Yaskawa INFORM job: TWIN_FRONT_SEARCH_90ST-1_5340.JBI

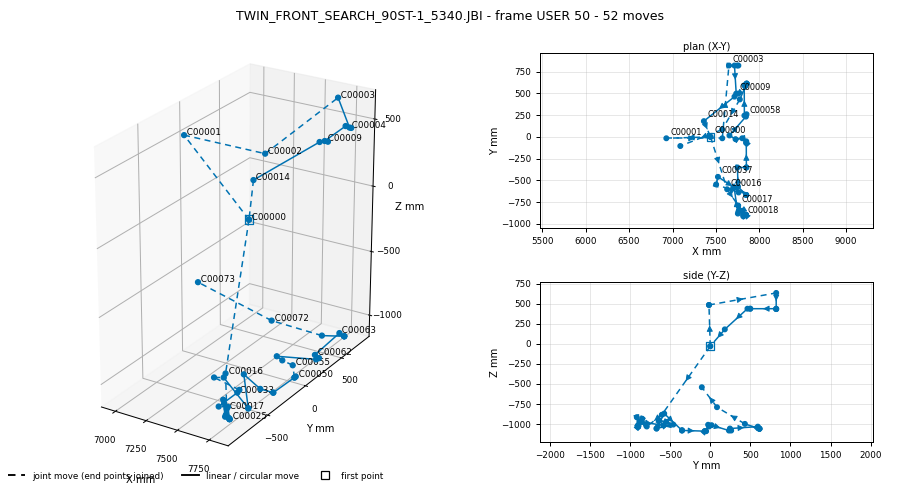
[picture p0: tool path of TWIN_FRONT_SEARCH_90ST-1_5340.JBI in frame USER 50, 52 of 56 moves have a stored position in this frame; points joined in program order, loops and branches not executed]
/JOB
//NAME TWIN_FRONT_SEARCH_90ST-1_5340
///FOLDERNAME 02-SKRZYNIE_JOBS
//POS
///NPOS 74,74,0,10,0,0
///USER 50
///TOOL 0
///POSTYPE USER
///RECTAN
///RCONF 0,0,1,0,0,0,0,0,0,0,0,0,0,0,0,0,0,0,0,0,0,0,0,0
C00000=7437.393,0.308,-30.113,-0.0036,-53.6521,0.0034
///RCONF 1,0,1,0,0,0,0,0,0,0,0,0,0,0,0,0,0,0,0,0,0,0,0,0
C00001=6928.400,-15.669,483.666,2.7707,-42.5282,-1.8493
C00002=7572.625,-15.669,483.666,2.7707,-42.5282,-1.8493
C00003=7649.331,821.904,633.544,31.3308,-50.3097,5.8371
C00004=7744.036,821.924,432.600,31.3309,-50.3106,5.8382
C00005=7764.657,821.900,432.619,31.3298,-50.3131,5.8368
C00006=7758.075,821.902,432.614,31.3294,-50.3128,5.8375
C00007=7758.087,821.893,399.298,31.3287,-50.3132,5.8373
C00008=7713.156,821.903,437.297,31.3290,-50.3132,5.8374
C00009=7733.152,498.705,437.301,28.5621,-56.7278,8.0159
C00010=7764.512,498.715,437.279,28.5577,-56.7277,8.0212
C00011=7758.151,498.718,437.279,28.5586,-56.7273,8.0207
C00012=7758.152,498.721,398.863,28.5594,-56.7235,8.0206
C00013=7713.145,463.670,437.302,31.3284,-50.3136,5.8380
C00014=7360.642,181.544,179.903,-30.3084,-22.7119,47.7634
///RCONF 0,0,1,0,0,0,0,0,0,0,0,0,0,0,0,0,0,0,0,0,0,0,0,0
C00015=7437.393,0.308,-30.113,-0.0036,-53.6521,0.0034
///RCONF 0,0,0,0,0,0,0,0,0,0,0,0,0,0,0,0,0,0,0,0,0,0,0,0
C00016=7628.865,-602.935,-884.155,-14.6080,-23.9960,-22.0349
///RCONF 1,0,0,0,0,0,0,0,0,0,0,0,0,0,0,0,0,0,0,0,0,0,0,0
C00017=7755.981,-790.379,-1030.058,-1.3034,-14.2488,-53.7856
C00018=7814.982,-914.673,-915.183,-49.7301,36.0224,40.1931
C00019=7814.976,-893.416,-1010.060,-49.7313,36.0195,40.1889
C00020=7814.973,-903.090,-1020.024,-49.7309,36.0192,40.1886
C00021=7814.980,-919.884,-1020.010,-49.7305,36.0200,40.1893
///RCONF 0,0,0,0,0,0,0,0,0,0,0,0,0,0,0,0,0,0,0,0,0,0,0,0
C00022=7765.216,-847.521,-933.099,-41.9556,-3.8768,2.5162
C00023=7838.256,-897.742,-1022.780,33.2636,-28.1441,-95.3546
C00024=7838.227,-897.761,-1034.874,33.2614,-28.1452,-95.3536
C00025=7845.758,-897.726,-1031.582,33.2648,-28.1427,-95.3555
C00026=7845.758,-897.726,-1031.582,33.2648,-28.1427,-95.3555
C00027=7845.758,-897.726,-1031.582,33.2648,-28.1427,-95.3555
C00028=7845.758,-897.726,-1031.582,33.2648,-28.1427,-95.3555
C00029=7863.986,-897.727,-1031.592,33.2632,-28.1430,-95.3545
C00030=7803.420,-850.217,-974.308,33.2648,-28.1422,-95.3567
///RCONF 1,0,0,0,0,0,0,0,0,0,0,0,0,0,0,0,0,0,0,0,0,0,0,0
C00031=7813.345,-897.089,-897.203,54.9948,73.9690,-177.4313
C00032=7752.242,-882.487,-971.733,-38.0360,-24.7001,-17.6899
C00033=7709.308,-583.044,-1014.454,-8.5802,-15.4711,-34.3684
///RCONF 0,0,0,0,0,0,0,0,0,0,0,0,0,0,0,0,0,0,0,0,0,0,0,0
C00034=7760.363,-639.479,-954.196,-16.2283,58.5864,108.1042
///RCONF 1,0,0,0,0,0,0,0,0,0,0,0,0,0,0,0,0,0,0,0,0,0,0,0
C00035=7501.819,-547.461,-973.110,-40.0484,29.0713,48.7679
C00036=7849.163,-652.269,-1055.293,-36.7283,45.9336,63.6180
C00037=7522.707,-459.746,-1006.152,21.9891,-7.6328,-78.4767
///RCONF 0,0,0,0,0,0,0,0,0,0,0,0,0,0,0,0,0,0,0,0,0,0,0,0
C00038=7848.448,-668.635,-1055.276,-38.1211,38.1551,84.2772
C00039=7848.418,-668.637,-1070.622,-38.1202,38.1533,84.2760
C00040=7859.950,-668.642,-1067.637,-38.1207,38.1516,84.2738
C00041=7848.448,-668.635,-1055.276,-38.1211,38.1551,84.2772
///RCONF 1,0,0,0,0,0,0,0,0,0,0,0,0,0,0,0,0,0,0,0,0,0,0,0
C00042=7753.744,-572.921,-869.370,35.5853,8.2503,-84.4804
///RCONF 0,0,0,0,0,0,0,0,0,0,0,0,0,0,0,0,0,0,0,0,0,0,0,0
C00043=7760.219,-665.415,-840.606,-36.5266,43.0988,92.6871
C00044=7778.037,-351.548,-1078.962,-31.8373,42.1277,84.4329
C00045=7747.357,-351.554,-1078.963,-31.8382,42.1272,84.4305
///RCONF 1,0,0,0,0,0,0,0,0,0,0,0,0,0,0,0,0,0,0,0,0,0,0,0
C00046=7850.194,-351.548,-1078.962,-31.8375,42.1274,84.4323
C00047=7850.215,-351.581,-1093.915,-31.8403,42.1281,84.4282
C00048=7861.111,-351.581,-1090.949,-31.8408,42.1244,84.4218
C00049=7850.194,-351.548,-1078.962,-31.8375,42.1274,84.4323
C00050=7848.886,-51.045,-1088.766,-31.8328,42.1278,99.9917
C00051=7848.894,-68.663,-1088.753,-31.8329,42.1298,99.9929
C00052=7848.906,-68.683,-1101.493,-31.8343,42.1324,99.9922
C00053=7861.752,-68.689,-1098.467,-31.8340,42.1361,99.9970
C00054=7848.894,-68.663,-1088.753,-31.8329,42.1298,99.9929
C00055=7802.761,-15.645,-1029.914,-9.7407,56.5457,162.3768
///RCONF 0,0,0,0,0,0,0,0,0,0,0,0,0,0,0,0,0,0,0,0,0,0,0,0
C00056=7725.278,-25.980,-1008.468,-14.6300,-10.2329,22.0522
C00057=7655.312,16.758,-1013.968,36.3468,26.5568,-107.0138
///RCONF 1,0,0,0,0,0,0,0,0,0,0,0,0,0,0,0,0,0,0,0,0,0,0,0
C00058=7844.634,233.760,-1080.855,23.4698,44.5725,-116.2756
C00059=7851.838,260.958,-1080.540,23.4723,44.5715,-116.2716
C00060=7851.821,261.021,-1099.017,23.4678,44.5749,-116.2769
C00061=7860.953,261.032,-1096.049,23.4627,44.5753,-116.2825
C00062=7827.288,245.626,-1055.543,23.4731,44.5712,-116.2696
C00063=7825.305,593.191,-1032.010,10.4642,52.1554,-131.8432
C00064=7853.529,612.933,-1058.080,10.4637,52.1549,-131.8455
C00065=7853.595,612.880,-1072.989,10.4677,52.1564,-131.8443
C00066=7853.565,612.921,-1058.045,10.4627,52.1566,-131.8492
C00067=7868.536,612.906,-1058.021,10.4653,52.1574,-131.8467
C00068=7853.558,612.926,-1058.047,12.0695,52.4631,-119.3669
C00069=7853.529,635.104,-1058.094,12.7425,52.9997,-118.8215
C00070=7853.561,612.917,-1058.050,10.4623,52.1563,-127.3651
C00071=7774.620,431.852,-997.566,17.4286,48.8596,-123.7766
C00072=7570.947,84.363,-789.769,8.3295,54.7414,-178.0447
C00073=7089.401,-104.773,-541.114,-34.6747,-14.1850,36.1511
///RCONF 0,0,0,0,0,0,0,0,0,0,0,0,0,0,0,0,0,0,0,0,0,0,0,0
BC00000=5622.975
BC00001=5622.975
BC00002=6267.199
BC00003=6480.663
BC00004=6480.663
BC00005=6480.663
BC00006=6480.663
BC00007=6480.663
BC00008=6480.663
BC00009=6480.663
BC00010=6480.663
BC00011=6480.663
BC00012=6480.663
BC00013=6480.663
BC00014=6140.736
BC00015=5622.975
BC00016=6179.171
BC00017=6446.713
BC00018=6446.759
BC00019=6446.759
BC00020=6446.759
BC00021=6446.759
BC00022=6446.759
BC00023=6446.759
BC00024=6446.759
BC00025=6446.759
BC00026=6446.759
BC00027=6446.759
BC00028=6446.759
BC00029=6446.759
BC00030=6446.759
BC00031=6446.759
BC00032=6446.759
BC00033=6379.471
BC00034=6379.472
BC00035=6162.623
BC00036=6515.049
BC00037=6162.623
BC00038=6515.049
BC00039=6515.049
BC00040=6515.049
BC00041=6515.049
BC00042=6419.547
BC00043=6419.547
BC00044=6442.892
BC00045=6445.014
BC00046=6515.049
BC00047=6515.049
BC00048=6515.049
BC00049=6515.049
BC00050=6515.049
BC00051=6515.049
BC00052=6515.049
BC00053=6515.049
BC00054=6515.049
BC00055=6439.422
BC00056=6439.422
BC00057=6307.353
BC00058=6515.049
BC00059=6515.049
BC00060=6515.049
BC00061=6515.049
BC00062=6515.049
BC00063=6515.029
BC00064=6515.029
BC00065=6515.035
BC00066=6515.035
BC00067=6515.035
BC00068=6515.035
BC00069=6515.035
BC00070=6515.035
BC00071=6515.035
BC00072=6132.885
BC00073=5388.459
///POSTYPE BASE
P00006=-2.449,0.031,8.825,0.0000,0.0000,0.0000
P00021=6.550,-0.003,-5.735,0.0000,0.0000,0.0000
P00022=5.943,-0.018,-6.388,0.0000,0.0000,0.0000
P00058=0.000,0.000,3.000,0.0000,0.0000,0.0000
///RCONF 1,0,0,0,0,0,0,0,0,0,0,0,0,0,0,0,0,0,0,0,0,0,0,0
P00500=2.332,-5.281,-1.258,0.0000,0.0000,0.0000
///RCONF 0,0,0,0,0,0,0,0,0,0,0,0,0,0,0,0,0,0,0,0,0,0,0,0
P00501=-2.026,0.009,3.534,0.0000,0.0000,0.0000
///RCONF 1,0,0,0,0,0,0,0,0,0,0,0,0,0,0,0,0,0,0,0,0,0,0,0
P00502=-2.023,0.001,1.732,0.0000,0.0000,0.0000
P00503=0.138,-0.044,1.539,0.0000,0.0000,0.0000
P00504=-0.309,-0.010,1.636,0.0000,0.0000,0.0000
P00505=0.999,-9.916,8.214,0.0000,0.0000,0.0000
//INST
///DATE 2025/01/21 12:44
///ATTR SC,RW,RJ
////FRAME USER 50
///GROUP1 RB1,BS1
NOP
MOVJ C00000 BC00000 VJ=50.00
MOVJ C00001 BC00001 VJ=50.00
MOVJ C00002 BC00002 VJ=50.00
MOVJ C00003 BC00003 VJ=50.00
MOVL C00004 BC00004 V=166.7
REFP 3 C00005 BC00005
CALL JOB:SEARCH-R1
SET P0021 P0006
SFTON P0021
MOVL C00006 BC00006 V=333.3 PL=0
REFP 3 C00007 BC00007
CALL JOB:SEARCH-R1
SET P0021 P0006
SFTON P0021
SFTOF
MOVL C00008 BC00008 V=166.7
MOVL C00009 BC00009 V=166.7
REFP 3 C00010 BC00010
CALL JOB:SEARCH-R1
SET P0022 P0006
SFTON P0022
MOVL C00011 BC00011 V=333.3 PL=0
REFP 3 C00012 BC00012
CALL JOB:SEARCH-R1
SET P0022 P0006
SFTON P0022
SFTOF
MOVL C00013 BC00013 V=166.7
MOVL C00014 BC00014 V=333.3
MOVJ C00015 BC00015 VJ=50.00
MOVJ C00016 BC00016 VJ=50.00
MOVJ C00017 BC00017 VJ=30.00
MOVJ C00018 BC00018 VJ=20.00
'::::::::::::::::::::::::::::::::
'W21 P
'::::::::::::::::::::::::::::::::
MOVL C00019 BC00019 V=500.0
MOVL C00020 BC00020 V=333.3 PL=0
REFP 3 C00021 BC00021
CALL JOB:SEARCH-R1
SET P0500 P0006
SFTON P0500
MOVL C00022 BC00022 V=333.3 PL=0
MOVL C00023 BC00023 V=333.3
REFP 3 C00024 BC00024
CALL JOB:SEARCH-R1
SET P0500 P0006
SFTON P0500
MOVL C00025 BC00025 V=333.3 PL=0
MOVL C00026 BC00026 V=333.3
MOVL C00027 BC00027 V=333.3
MOVL C00028 BC00028 V=333.3
REFP 3 C00029 BC00029
CALL JOB:SEARCH-R1
SET P0500 P0006
SFTOF
MOVL C00030 BC00030 V=166.7
COMM MOVL C00031 BC00031 V=166.7
MOVJ C00032 BC00032 VJ=30.00
MOVL C00033 BC00033 V=333.3
'::::::::::::::::::::::::::::::::
'W21 L
'::::::::::::::::::::::::::::::::
MOVJ C00034 BC00034 VJ=30.00
MOVJ C00035 BC00035 VJ=30.00
COMM MOVL C00036 BC00036 V=333.3
MOVJ C00037 BC00037 VJ=30.00
MOVL C00038 BC00038 V=333.3 PL=0
REFP 3 C00039 BC00039
CALL JOB:SEARCH-R1
IMOV P0058 V=16.7
SET P0501 P0006
SFTON P0501
REFP 3 C00040 BC00040
CALL JOB:SEARCH-R1
SET P0501 P0006
SFTON P0501
MOVL C00041 BC00041 V=500.0 PL=0
SFTOF
'::::::::::::::::::::::::::::::::
'W20 P
'::::::::::::::::::::::::::::::::
MOVL C00042 BC00042 V=250.0
COMM MOVL C00043 BC00043 V=166.7
COMM MOVL C00044 BC00044 V=333.3
MOVL C00045 BC00045 V=333.3
MOVL C00046 BC00046 V=333.3 PL=0
REFP 3 C00047 BC00047
CALL JOB:SEARCH-R1
IMOV P0058 V=16.7
SET P0502 P0006
SFTON P0502
REFP 3 C00048 BC00048
CALL JOB:SEARCH-R1
SET P0502 P0006
SFTON P0502
MOVL C00049 BC00049 V=500.0 PL=0
SFTOF
'::::::::::::::::::::::::::::::::
'W20 L
'::::::::::::::::::::::::::::::::
MOVL C00050 BC00050 V=250.0
MOVL C00051 BC00051 V=333.3 PL=0
REFP 3 C00052 BC00052
CALL JOB:SEARCH-R1
IMOV P0058 V=16.7
SET P0503 P0006
SFTON P0503
REFP 3 C00053 BC00053
CALL JOB:SEARCH-R1
SET P0503 P0006
SFTON P0503
MOVL C00054 BC00054 V=500.0 PL=0
SFTOF
'::::::::::::::::::::::::::::::::
'W22 P
'::::::::::::::::::::::::::::::::
MOVJ C00055 BC00055 VJ=30.00
MOVJ C00056 BC00056 VJ=30.00
MOVL C00057 BC00057 V=333.3
MOVL C00058 BC00058 V=333.3
MOVL C00059 BC00059 V=333.3 PL=0
REFP 3 C00060 BC00060
CALL JOB:SEARCH-R1
IMOV P0058 V=16.7
SET P0504 P0006
SFTON P0504
REFP 3 C00061 BC00061
CALL JOB:SEARCH-R1
SET P0504 P0006
SFTON P0504
MOVL C00062 BC00062 V=500.0 PL=0
SFTOF
'::::::::::::::::::::::::::::::::
'W22 L
'::::::::::::::::::::::::::::::::
MOVL C00063 BC00063 V=333.3
MOVL C00064 BC00064 V=333.3 PL=0
REFP 3 C00065 BC00065
CALL JOB:SEARCH-R1
SET P0505 P0006
SFTON P0505
MOVL C00066 BC00066 V=333.3 PL=0
REFP 3 C00067 BC00067
CALL JOB:SEARCH-R1
SET P0505 P0006
SFTON P0505
MOVL C00068 BC00068 V=333.3 PL=0
REFP 3 C00069 BC00069
CALL JOB:SEARCH-R1
SET P0505 P0006
SFTOF
MOVL C00070 BC00070 V=83.3
MOVL C00071 BC00071 V=333.3
MOVJ C00072 BC00072 VJ=40.00
MOVJ C00073 BC00073 VJ=80.00
END
